SUBAPPLICATION PAGES (* Subapplication Type *)
  (* Standard: 61499-2 *)
  (* Version 1.0, 2023-02-06, franz *)
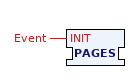
  EVENT_INPUT
    INIT;
  END_EVENT
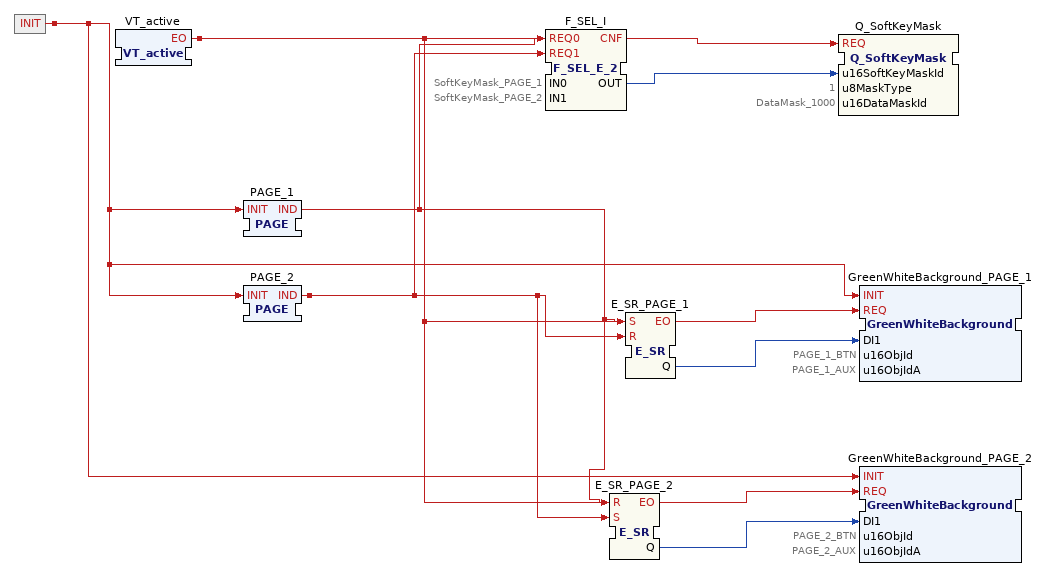
  FBS
    Q_SoftKeyMask : Q_SoftKeyMask(u8MaskType := 1, u16DataMaskId := DataMask_1000);
    F_SEL_I : F_SEL_E_2(IN0 := SoftKeyMask_PAGE_1, IN1 := SoftKeyMask_PAGE_2);
    E_SR_PAGE_1 : E_SR;
    E_SR_PAGE_2 : E_SR;
  END_FBS
  SUBAPPS
    VT_active : VT_active;
    GreenWhiteBackground_PAGE_2 : GreenWhiteBackground(u16ObjId := PAGE_2_BTN, u16ObjIdA := PAGE_2_AUX);
    GreenWhiteBackground_PAGE_1 : GreenWhiteBackground(u16ObjId := PAGE_1_BTN, u16ObjIdA := PAGE_1_AUX);
    PAGE_1 : PAGE;
    PAGE_2 : PAGE;
  END_SUBAPPS
  EVENT_CONNECTIONS
    F_SEL_I.CNF TO Q_SoftKeyMask.REQ;
    VT_active.EO TO F_SEL_I.REQ0;
    VT_active.EO TO E_SR_PAGE_1.S;
    VT_active.EO TO E_SR_PAGE_2.R;
    INIT TO GreenWhiteBackground_PAGE_2.INIT;
    E_SR_PAGE_2.EO TO GreenWhiteBackground_PAGE_2.REQ;
    INIT TO GreenWhiteBackground_PAGE_1.INIT;
    E_SR_PAGE_1.EO TO GreenWhiteBackground_PAGE_1.REQ;
    INIT TO PAGE_1.INIT;
    PAGE_1.IND TO F_SEL_I.REQ0;
    PAGE_1.IND TO E_SR_PAGE_1.S;
    PAGE_1.IND TO E_SR_PAGE_2.R;
    INIT TO PAGE_2.INIT;
    PAGE_2.IND TO F_SEL_I.REQ1;
    PAGE_2.IND TO E_SR_PAGE_2.S;
    PAGE_2.IND TO E_SR_PAGE_1.R;
  END_CONNECTIONS
  DATA_CONNECTIONS
    F_SEL_I.OUT TO Q_SoftKeyMask.u16SoftKeyMaskId;
    E_SR_PAGE_2.Q TO GreenWhiteBackground_PAGE_2.DI1;
    E_SR_PAGE_1.Q TO GreenWhiteBackground_PAGE_1.DI1;
  END_CONNECTIONS
END_SUBAPPLICATION
